(* IEC 61131-3 sources: SmartHomeNew/SmartHomeNew-main/workspace/system_layer_cleanup/comparison/shadow_outputs, 1 file *)

(* ---- FB_CoreKernel_Shadow_Outputs_DRAFT.st ---- *)
FUNCTION_BLOCK FB_CoreKernel_Shadow_Outputs_DRAFT
VAR_INPUT
    VI_Shadow_Path_Ready : BOOL;
END_VAR
VAR_OUTPUT
    VO_Shadow_Path_Ready : BOOL;
END_VAR

VO_Shadow_Path_Ready := VI_Shadow_Path_Ready;

END_FUNCTION_BLOCK
